FUNCTION_BLOCK FB_LightPIR
VAR_INPUT
	bInputPIR		:	BOOL;						//Input des Bewegungsmelders
	bInputSecLoop	:	BOOL := FALSE;				//Input für Security Loop
	tHigh			:	TIME;						//Zeit (ms) für High
END_VAR
VAR_IN_OUT
	bInputHA		:	BOOL;						//Input (HA)
END_VAR
VAR_OUTPUT
	bOut			:	BOOL;
END_VAR
VAR CONSTANT
	tSec			:	TIME := T#1S;
END_VAR
VAR
	fbRtrigPIR		:	R_TRIG;
	fbTrigSec		:	R_TRIG;
	
	bStateOut		:	BOOL := FALSE;

	tpPulse			:	TP_RST;
	
	tpPulseSec		:	TP;
	tofDelaySec		:	TOF;
END_VAR

// Security Loop
fbTrigSec	(CLK:= bInputPIR, Q=> );

IF bInputSecLoop THEN
	
	tpPulseSec	(IN := bStateOut, PT := tSec);
    tofDelaySec	(IN := bStateOut, PT := tSec);

	IF fbTrigSec.Q THEN
		bStateOut	:= TRUE;
	END_IF
	
	IF NOT tpPulseSec.Q THEN
		bStateOut := FALSE;
	END_IF
	
	IF NOT tofDelaySec.Q THEN
		bStateOut := TRUE;
	END_IF	

ELSIF bInputHA THEN

	bStateOut := TRUE;

ELSE

	fbRtrigPIR(CLK:= bInputPIR, Q=> );
	
	// Pulse
	tpPulse(IN := fbRtrigPIR.Q, PT := tHigh);

	IF tpPulse.Q THEN
		bStateOut	:= TRUE;
		
		//Reset Pulse bei neuer erkennung
		tpPulse.RST := fbRtrigPIR.Q;
		
	ELSE
		bStateOut 	:= FALSE;
	END_IF
	
	IF bInputPIR THEN
		bStateOut	:= TRUE;
	END_IF

END_IF

bOut		:= bStateOut;

END_FUNCTION_BLOCK

(* stored: Version 1.1.0.1, ProductVersion 3.1.4024.4
   POU FB_LightPIR: Id {18fc6d29-bfc9-47ea-816f-b72b3250efe3}, SpecialFunc None *)
